{attribute 'GeneratedUsingTerminal: EP1809-0042-0018'}
{attribute addProperty BoxType "EP1809-0042-0018"}
{attribute addProperty Id "InputAT %I*BOOL1"}
{attribute addProperty CRC "2198356929"}
{attribute addProperty Size "1"}
TYPE DI_X01_Pin_830843C1 EXTENDS InputBase_8311D824 :
STRUCT
	{attribute addProperty Name "Input"}
	Input AT %I* : BOOL;
END_STRUCT
END_TYPE

(* stored: Version 1.2.0.0, ProductVersion 3.1.4024.11
   DUT DI_X01_Pin_830843C1: Id {91a8d2ec-acdd-4618-becf-59959f17b6ad} *)
